// TIA Portal V16 export
// export: Created 2022-09-01T13:37:27.0954718Z, ExportSetting WithDefaults, DisplayName Totally Integrated Automation Portal, DisplayVersion V16, DisplayName TIA Portal Version Control Interface, DisplayVersion V16, DisplayName TIA Portal Openness, DisplayVersion V16, DisplayName STEP 7 Professional, DisplayVersion V16, DisplayName STEP 7 Safety, DisplayVersion V16, DisplayName WinCC Advanced, DisplayVersion V16
VAR_GLOBAL   // PLC tag table "Saídas"
   BS001A AT %Q0.0 : Bool;
   BS001B AT %Q0.1 : Bool;
   XV101 AT %Q3.3 : Bool;
   XV102 AT %Q3.4 : Bool;
   MX201 AT %Q0.4 : Bool;
   BH201 AT %Q0.5 : Bool;
   MX301 AT %Q0.6 : Bool;
   ALIM_BM401 AT %Q0.7 : Bool;
   LIGAR_BM401 AT %Q3.1 : Bool;
   BS501 AT %Q1.1 : Bool;
   MX601 AT %Q2.0 : Bool;
   BD601 AT %Q2.1 : Bool;
   BD602 AT %Q2.2 : Bool;
   MX603 AT %Q2.3 : Bool;
   BD603 AT %Q2.4 : Bool;
   MX604 AT %Q2.5 : Bool;
   BD604 AT %Q2.6 : Bool;
   MX605 AT %Q2.7 : Bool;
   BD605 AT %Q0.2 : Bool;
   ALARME AT %Q3.2 : Bool;
END_VAR
